(* Logix 5000 project; controller Transcat vendor 1 type 14 code 152 rev 32.11; software revision 32.02 *)

TASK MainTask (continuous, watchdog 500 ms) : MainProgram

MODULES
   Local : vendor 1 type 14 code 152 (PointIO 0, rev 32.11)
      MX201_LowerHowesVFD : PowerFlex 525-EENET (Ethernet 192.168.1.192, rev 5.1, Output RPI 20 ms)   // VFD for Lower Howes Mixer
           MX201_LowerHowesVFD:I.Ready   // LowerHowes Drive Ready Status
           MX201_LowerHowesVFD:I.Faulted   // LowerHowes Drive Faulted
           MX201_LowerHowesVFD:I.Active   // LowerHowes Drive Active
           MX201_LowerHowesVFD:O.Stop   // Drive Stop
      MX101_UpperHowesVFD : PowerFlex 525-EENET (Ethernet 192.168.1.191, rev 5.1, Output RPI 20 ms)   // VFD for Upper Howes Mixer
           MX101_UpperHowesVFD:I.Faulted   // UpperHowes Drive Faulted
           MX101_UpperHowesVFD:I.Active   // UpperHowes Drive Active
           MX101_UpperHowesVFD:I.Ready   // UpperHowes Drive Ready Status
           MX101_UpperHowesVFD:O.FreqCommand   // Input Hz into Source A: 0-60 Hz range
           MX101_UpperHowesVFD:O.Stop   // Drive Stop
           MX101_UpperHowesVFD:O.Start   // Drive Start
      VF101_Medium_Feeder : PowerFlex 525-EENET (Ethernet 192.168.1.193, rev 5.1, Output RPI 20 ms)   // Medium Feeder
      VF201_Small_Feeder_2 : PowerFlex 525-EENET (Ethernet 192.168.1.194, rev 5.1, Output RPI 20 ms)   // Small Feeder 2
      Thayer1_BS : ETHERNET-MODULE (Ethernet 192.168.1.140, rev 1.1, Output RPI 50 ms)   // Thayer 1 Weight Belt Feeder
      SBC2000_1_Acrison : ETHERNET-MODULE (Ethernet 192.168.1.150, rev 1.1, Output RPI 250 ms)   // Acrison Drive 1 to control Small Feeder 1
           SBC2000_1_Acrison:I.Data[1]   // PV - Feedrate - kg/hr
           SBC2000_1_Acrison:I.Data[2]   // Totalizer 1 - kg
           SBC2000_1_Acrison:I.Data[4]   // Hopper Level - %
           SBC2000_1_Acrison:I.Data[3]   // OT - Motor Speed - %
           SBC2000_1_Acrison:I.Data   // Ethernet Input Array
           SBC2000_1_Acrison:I.Data[0]   // SP-FeedRate - kg/hr
           SBC2000_1_Acrison:O.Data[15]   // When Command_Bits is 1, machine is running.
      Thayer2_BS : ETHERNET-MODULE (Ethernet 192.168.1.160, rev 1.1, Output RPI 50 ms)   // Thayer 2 Weigh Belt Feeder
      AENTPointIO : 1734-AENT (Ethernet 192.168.1.190, rev 3.1, Output RPI 20 ms)
         Slot1_420_8Input : vendor 1 type 115 code 210 (PointIO 1, rev 3.1, Input RPI 80 ms)
              AENTPointIO:1:I.Ch0Data   // LowerHowesSpeedSensorSignal
         Slot2_24V_8DI : 1734-IB8 (PointIO 2, rev 3.1)
      Discrete_IO : Embedded (PointIO 1, rev 32.11, Output RPI 20 ms)
           Local:1:O.Data.0   // Red Beacon Light
           Local:1:O.Data.3   // Blue Beacon Light
           Local:1:O.Data.1   // Yellow Beacon Light
           Local:1:O.Data.2   // Green Beacon Light
           Local:1:O.Data.4   // Beacon Buzzer/Sound
END_MODULES

TYPE Acrison_Feeder :   // Acrison Feeder Tags
STRUCT
   AutoMan : BOOL;   // On - Auto Control - follows AutoRun bit, Off - Manaul Control - follows Manual Run bit
   ManualRun : BOOL;   // On - Runs feeder in Manual, Off - Stops feeder in manual
   AutoRun : BOOL;   // On - Runs feeder in Auto Off - Stops feeder in Auto
   Interlock : BOOL;   // Interlock bit - if on - Feeder will not run
   Output : BOOL;   // On - Feeder runs, Off Feeder stops
   Int_Status : DINT;   // 32 Status bits from feeder
   SP_HMI : REAL;   // setpoint from HMI
   SP_READ : REAL;   // setpoint read back from controller
   Enable : BOOL;   // Enable logic to run feeder
   OT_Actual_Hz : REAL;   // The current output of the VFD in Hz
   FreqHz_Real : REAL;   // The command frequency of the drive in Hz
   CycleTime : TIMER;   // running time of current cycle
   CampTime : TIMER;   // running time of current campaign / batch
   TotalTime : TIMER;   // total time the device / motor has run since last reset
   OneShots : BOOL[32];   // 32 Booleans to hold one-shots assicated with this device
   TimeRunTarget : DINT;   // Target Amount of time in seconds to run the device
   StartDelay : TIMER;   // Delay before motor start
   StartDelayms : DINT;   // Start delay in milliseconds
   TimeRunStart : BOOL;   // Bit to start and run a timed run
END_STRUCT
END_TYPE

TYPE BronkhorstFlowMeter :   // Read and write values for Bronkhorst Flow Meters
STRUCT
   SP_R : REAL;   // Set Point - FlowRate - Read - g/min - read from Flow Meter
   PV_R : REAL;   // Process Variable - FlowRate - Read - g/min
   OT_R : REAL;   // Output - PumpSpeed - Read - %
   TempC : REAL;   // Temperaure - Read - Deg C
   Density : REAL;   // Density - Read - g/liter
   Usertag : STRING;   // User Tag in Flow Meter - String
   FBNode : INT;   // Flow Bus Node # - Integer
   Model : STRING;   // Flow Meter Model #
   Serial : STRING;   // Flow Meter Serial #
   Capacity : REAL;   // Max Flow Rate of Flow Meter
   Enable : BOOL;   // Device enable bit
   AutoMan : BOOL;   // Select Auto / Manual Mode
   AutoRun : BOOL;   // On / Off in Auto Mode
   ManualRun : BOOL;   // On / Off- in Manual Mode
   Interlock : BOOL;   // Interlock Bit
   Output : BOOL;   // Output Bit for Device
   SP_HMI : REAL;   // Setpoint from HMI
   SP_W : REAL;   // Setpoint - flowrate g/min - write to Flow Meter from PLC
   Connected : BOOL;   // Is flow meter connecte to the flow bus network
   Alarm : BOOL;   // Alarm Bit - if on flow meter in ALarm Status
   Running : BOOL;   // the flow meter is running / dosing
   AlarmReset : BOOL;   // bit to toggle to reset alarm
   AlarmID : INT;   // Integer # that describes the type of Alarm
   ReadTime : INT;   // time in milliseconds to read the flow meter data
   DevPct : REAL;   // % deviation of process variable from setpoint
   CycleTime : TIMER;   // running time of current cycle
   CampTime : TIMER;   // running time of current campaign
   TotalTime : TIMER;   // total time the device / motor has run since last reset
   OneShots : BOOL[32];   // 32 Booleans to hold one-shots assicated with this device
   TimeRunTarget : DINT;   // Target Amount of time in seconds to run the device
   StartDelay : TIMER;   // Delay before motor start
   StartDelayms : DINT;   // Start delay in milliseconds
   TimeRunStart : BOOL;   // Bit to start and run a timed run
END_STRUCT
END_TYPE

TYPE Howes_Mixer :   // Howes Mixer Tags
STRUCT
   AutoMan : BOOL;   // On - Auto Control - follows AutoRun bit, Off - Manaul Control - follows Manual Run bit
   ManualRun : BOOL;   // On - Runs feeder in Manual, Off - Stops feeder in manual
   AutoRun : BOOL;   // On - Runs feeder in Auto Off - Stops feeder in Auto
   Interlock : BOOL;   // Interlock bit - if on - Feeder will not run
   Output : BOOL;   // On - Feeder runs, Off Feeder stops
   Int_Status : DINT;   // 32 Status bits from feeder
   SP_HMI : REAL;   // setpoint from HMI
   SP_READ : REAL;   // setpoint read back from controller
   Enable : BOOL;   // Enable logic to run mixer
   FreqHz_Real : REAL;   // Frequency in Hz expressed as real #
   OT_Actual_Hz : REAL;   // The current output of the drive in Hz
   CycleTime : TIMER;   // currnet cycle run time
   CampTime : TIMER;   // current campaign run time
   TotalTime : TIMER;   // total run time since last reset
   OneShots : BOOL[32];   // 32 Booleans to hold one shots associated with this device
   TimeRunTarget : DINT;   // Target Amount of time in seconds to run the device
   TimeRunStart : BOOL;   // Bit to start and run a timed run
   StartDelay : TIMER;   // Delay before motor starts
   StartDelayms : DINT;   // Delay before motor starts in milliseconds
   RPM : REAL;   // RPM from speed sensor
END_STRUCT
END_TYPE

TYPE Thayer_WB_Feeder :   // Thayer WB Feeder Tags
STRUCT
   AutoMan : BOOL;   // On - Auto Control - follows AutoRun bit, Off - Manaul Control - follows Manual Run bit
   ManualRun : BOOL;   // On - Runs feeder in Manual, Off - Stops feeder in manual
   AutoRun : BOOL;   // On - Runs feeder in Auto Off - Stops feeder in Auto
   Interlock : BOOL;   // Interlock bit - if on - Feeder will not run
   Output : BOOL;   // On - Feeder runs, Off Feeder stops
   Int_Status : DINT;   // 32 Status bits from feeder
   SP_HMI : REAL;   // setpoint from HMI
   SP_READ : REAL;   // setpoint read back from controller
   Enable : BOOL;   // Enable logic to run feeder
   CycleTime : TIMER;   // current cycle run time
   CampTime : TIMER;   // current campaing run time
   TotalTime : TIMER;   // total run time since last reset
   OneShots : BOOL[32];   // 32 Booleans to hold one-shots assicated with this device
   TimeRunTarget : DINT;   // Target Amount of time in seconds to run the device - from recipe
   StartDelay : TIMER;   // Delay before starting motor / equipment
   StartDelayms : DINT;   // Start delay in milliseconds
   TimeRunStart : BOOL;   // Bit to start and run a timed run
END_STRUCT
END_TYPE

VAR_GLOBAL   (* controller tags *)
   AcrisonFeedRateSetPoint : MESSAGE;   // Message Command to Write to Feed Rate Set Point in Acrison from GF103.SP_HMI in kg/hr
        MessageParameters(ServiceCode := 16#0010, LocalElement := GF301.SP_HMI, ...)
   alwaysOFF : BOOL := 1;
   BeaconBeepAlarm : ALIAS FOR Local:1:O.Data.4;   // Beep Alarm
   BeaconBlueLight : ALIAS FOR Local:1:O.Data.3;   // Blue Beacon Light
   BeaconGreenLight : ALIAS FOR Local:1:O.Data.2;   // Green Beacon Light
   BeaconRedLight : ALIAS FOR Local:1:O.Data.0;   // Red Beacon Light
   BeaconYellowLight : ALIAS FOR Local:1:O.Data.1;   // Yellow Beacon Light
   Beep : BOOL;   // Bit to Activte Beacon Alarm
   FT103 : BronkhorstFlowMeter := (PV_R := -36.801758, TempC := 22.806396, Density := 9999.0, Usertag := 'FT-103', Model := 'M55-RGD-25-0-S', Serial := 'M22213015A', Capacity := 1000.00006, Enable := 1, SP_HMI := 45.67, Connected := 1, Alarm := 1, AlarmID := 40, ReadTime := 72, CycleTime.PRE := 288000000, CycleTime.ACC := 5305, CampTime.PRE := 28800000, CampTime.ACC := 10001, TotalTime.PRE := 999999999, TotalTime.ACC := 47616, StartDelay.PRE := 1000, StartDelayms := 1);
   FT104 : BronkhorstFlowMeter := (PV_R := -6.675215, TempC := 22.177925, Density := 9999.0, Usertag := 'FT-104          ', Model := 'M55-RGD-25-0-S', Serial := 'M22213015C', Capacity := 10000.0, Enable := 1, SP_HMI := 100.0, Connected := 1, ReadTime := 95, CycleTime.PRE := 288000000, CycleTime.ACC := 4100, CampTime.PRE := 28800000, CampTime.ACC := 10001, TotalTime.PRE := 999999999, TotalTime.ACC := 72384, StartDelay.PRE := 2000, StartDelayms := 2);
   FT105 : BronkhorstFlowMeter := (PV_R := 0.5933827, TempC := 29.03157, Density := 4.8631186, Usertag := 'FT-105          ', Model := 'M14-RGD-22-0-S', Serial := 'M20210127A', Capacity := 202.79999, Enable := 1, SP_HMI := 56.78, Connected := 1, ReadTime := 63, CycleTime.PRE := 288000000, CycleTime.ACC := 5050, CampTime.PRE := 28800000, CampTime.ACC := 10001, TotalTime.PRE := 999999999, TotalTime.ACC := 27737, StartDelay.PRE := 4000, StartDelayms := 4);
   GF101 : Thayer_WB_Feeder := (SP_HMI := 14.7, SP_READ := 14.6875, Enable := 1, CycleTime.PRE := 288000000, CycleTime.ACC := 2365, CampTime.PRE := 28800000, CampTime.ACC := 10001, TotalTime.PRE := 999999999, TotalTime.ACC := 1588506, StartDelay.PRE := 5000, StartDelayms := 5);   // Thayer 1 Tags
   GF201 : Thayer_WB_Feeder := (SP_HMI := 12.5, SP_READ := 12.5, Enable := 1, CycleTime.PRE := 288000000, CycleTime.ACC := 9602, CampTime.PRE := 28800000, CampTime.ACC := 10001, TotalTime.PRE := 999999999, TotalTime.ACC := 1608497, StartDelay.PRE := 3000, StartDelayms := 3);   // Thayer 2 Tags
   GF301 : Acrison_Feeder := (Int_Status := 591964, SP_HMI := 5.0, Enable := 1, CycleTime.PRE := 288000000, CycleTime.ACC := 6447, CampTime.PRE := 28800000, CampTime.ACC := 10001, TotalTime.PRE := 999999999, TotalTime.ACC := 1606494, StartDelay.PRE := 2000, StartDelayms := 2);   // GF103 - Small Feeder 1
        .Int_Status.11   // Alarm
        .Int_Status.13   // Empty
        .Int_Status.10   // Overfill / Empty
        .Int_Status.3   // SP Int-1 / Ext-0
        .Int_Status   // 32 Bit Status Int
        .Int_Status.0   // Run-1 / Stop-0
        .Int_Status.5   // Batch-1 / Cont-0
        .Int_Status.4   // Mode - Grav-1 / Vol-0
        .Int_Status.6   // Batch Complete
        .Int_Status.1   // Refil
        .Int_Status.7   // Bribble
        .Int_Status.12   // Message
        .Int_Status.9   // Low Level
        .Int_Status.14   // Overfill
        .Int_Status.15   // Acrilock
        .Int_Status.16   // No Scale
        .Int_Status.17   // Deviation
        .Output   // GF103 - Acrison Small Feeder Run Bit
        .Int_Status.2   // AutoRefill
        .Int_Status.8   // High Level
   GreenFlashingOff : TIMER := (PRE := 500);
   GreenFlashingOn : TIMER := (PRE := 500);
   HertzSetting : ALIAS FOR MX101_UpperHowesVFD:O.FreqCommand.0;   // UserHzSetting
   MSG_FROM_SLC500 : INT[10] := ([1] := 2500, [2] := 200, [3] := 300, [4] := 400, [5] := 500, [6] := 16, [7] := 17, [8] := 18, [9] := 19); {produced}
   MX101 : Howes_Mixer := (SP_HMI := 5.0, Enable := 1, FreqHz_Real := 3.0, CycleTime.PRE := 288000000, CycleTime.ACC := 3118, CampTime.PRE := 28800000, CampTime.ACC := 10001, TotalTime.PRE := 999999999, TotalTime.ACC := 1718665, StartDelay.PRE := 5000, StartDelayms := 5);
   MX201 : Howes_Mixer := (SP_HMI := 10.0, Enable := 1, FreqHz_Real := 6.0, CycleTime.PRE := 28800000, CycleTime.ACC := 7089, CampTime.PRE := 28800000, CampTime.ACC := 10001, TotalTime.PRE := 999999999, TotalTime.ACC := 835800, StartDelay.PRE := 2000, StartDelayms := 2, RPM := -0.04);
   PowerOffThayer1 : BOOL;
   PowerOnThayer1 : BOOL;
   RandomFloat : REAL[20] := ([1] := 7.316811, [2] := 20.713356, [3] := 16.079597, [4] := 74.3938, [5] := 86.28061, [6] := 69.73996, [7] := 47.361, [8] := 43.876316, [9] := 89.62069, [10] := 56.526745);
   RecipeStart : BOOL;   // Bit to start and stop a recipe execution
   StartBeepTimer : TIMER := (PRE := 2500);   // Timer to sound the beep alarm before starting a device
   TempReal1 : REAL;
   Thayer1_SP : REAL := 20.0;
   Thayer1Ackn_SilenceRequest : BOOL;
   Thayer1Automatic : BOOL;
   Thayer1Data : REAL[40] := ([0] := -0.072265625, [1] := 4.6216e-41, [3] := 14.6875, [4] := 2.0, [9] := -0.19335938, [10] := -0.19343926, [11] := 7.512e-42, [15] := -0.071777344, [16] := 70.84617, [17] := 1.6071e-41, [19] := -0.072265625);
        [10]   // Totalizer 2
        [3]   // SetPoint
        [2]   // Running Speed
        [0]   // Running Load
        [1]   // Running Rate
        [9]   // Totalizer 1
   Thayer1PowerOn : BOOL;
   Thayer1ResetTotalizers : BOOL;
   Thayer1SetPoint : REAL[1];
   Thayer1SpeedControl : REAL := 20.0;
   Thayer2_SP : REAL := 20.0;
   Thayer2Automatic : BOOL;
   Thayer2Data : REAL[40] := ([0] := 3.609375, [1] := 7.6406e-41, [3] := 12.5, [15] := 3.609375, [16] := 70.91538, [17] := 1.6071e-41, [19] := 3.609375);
   Thayer2PowerOn : BOOL;
   Thayer2ResetTotalizers : BOOL;
   Thayer2SpeedControl : REAL := 20.0;
   UHStartOneShot : BOOL;
   UHStopOneShot : BOOL;
   UpHowesHMIRun : BOOL;
   UpHowesHMIStop : BOOL;
   UpHowesSpeedHMI : INT;
   UpperHowesSpeed : INT := 2500;
   UpperHowesStart : BOOL;
   UpperHowesStop : BOOL;
   VF101 : Acrison_Feeder := (SP_HMI := 10.0, Enable := 1, FreqHz_Real := 6.0, CycleTime.PRE := 288000000, CycleTime.ACC := 7359, CampTime.PRE := 28800000, CampTime.ACC := 10001, TotalTime.PRE := 999999999, TotalTime.ACC := 1720239, StartDelay.PRE := 5000, StartDelayms := 5);   // Medium Feeder Tags
   VF201 : Acrison_Feeder := (SP_HMI := 10.0, Enable := 1, FreqHz_Real := 6.0, CycleTime.PRE := 288000000, CycleTime.ACC := 13534, CampTime.PRE := 28800000, CampTime.ACC := 10001, TotalTime.PRE := 999999999, TotalTime.ACC := 1964985, StartDelay.PRE := 5000, StartDelayms := 5);   // Small Feeder 2 Tags
   YellowFlashOff : TIMER := (PRE := 500);
   YellowFlashOn : TIMER := (PRE := 500);
END_VAR

PROGRAM MainProgram   (* main routine MainRoutine *)
VAR
   AcrisonSpeedControl : REAL := 1.0;
   AcrisonSpeedControl2 : REAL := 15.0;
   Command_Bits : INT;
        .0   // GF103 - Acrison Small Feeder 1 - Run/Stop
   HertzInput : INT := 20;
   Int_Status : DINT := 540252;
   LowerHowesSpeedSensor : REAL := -74.39945;
   PowerOffACrison : BOOL := 1;
   PowerOnAcrison : BOOL;
   SCL_01 : SCALE := (In := -3.0, InRawMax := 16384.0, InRawMin := 3271.0, InEUMax := 300.0, Out := -74.90277, MinAlarm := 1);
   SCL_02 : SCALE := (In := 19.0, InRawMax := 16384.0, InRawMin := 3271.0, InEUMax := 300.0, Out := -74.39945, MinAlarm := 1);
   SpeedSensorUpperHowesSpeed : REAL := -74.90277;
   T1 : TIMER := (PRE := 10000);
   T2 : TIMER := (PRE := 10000, ACC := 10000, EN := 1, DN := 1);
END_VAR

ROUTINE FT103_Oil_Dosing   (* ladder *)
// Logic to control FT103
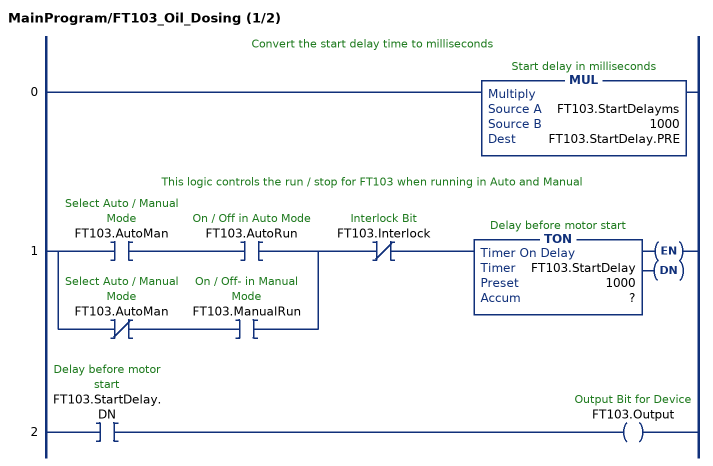
   // Convert the start delay time to milliseconds
   0: MUL(FT103.StartDelayms,1000,FT103.StartDelay.PRE);
   // This logic controls the run / stop for FT103 when running in Auto and Manual
   1: [XIC(FT103.AutoMan) XIC(FT103.AutoRun) ,XIO(FT103.AutoMan) XIC(FT103.ManualRun) ]XIO(FT103.Interlock)TON(FT103.StartDelay,?,?);
   2: XIC(FT103.StartDelay.DN)OTE(FT103.Output);
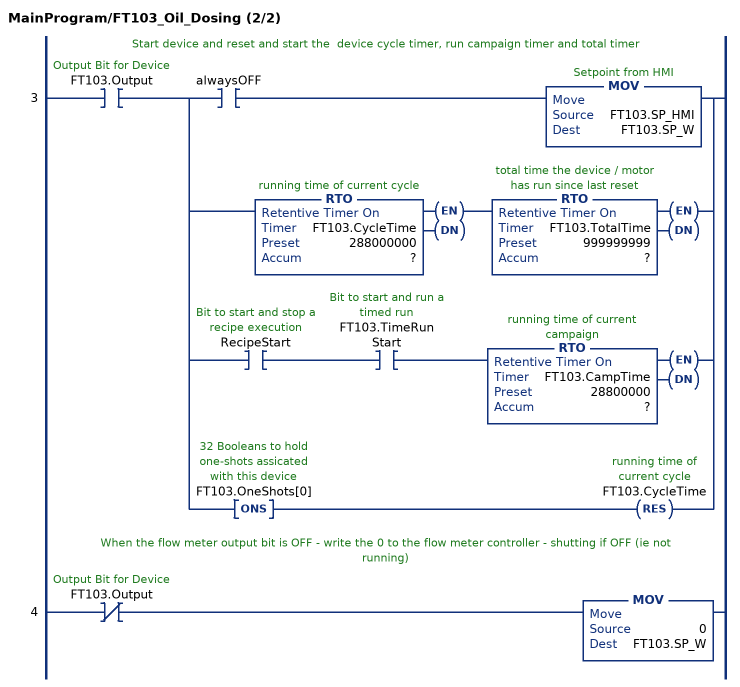
   // Start device and reset and start the  device cycle timer, run campaign timer and total timer
   3: XIC(FT103.Output)[XIC(alwaysOFF) MOV(FT103.SP_HMI,FT103.SP_W) ,[RTO(FT103.CycleTime,?,?) RTO(FT103.TotalTime,?,?) ,XIC(RecipeStart) XIC(FT103.TimeRunStart) RTO(FT103.CampTime,?,?) ,ONS(FT103.OneShots[0]) RES(FT103.CycleTime) ] ];
   // When the flow meter output bit is OFF - write the 0 to the flow meter controller - shutting if OFF (ie not running)
   4: XIO(FT103.Output)MOV(0,FT103.SP_W);
END_ROUTINE

ROUTINE FT104_Water_Dosing   (* ladder *)
// FT104 Control Logic
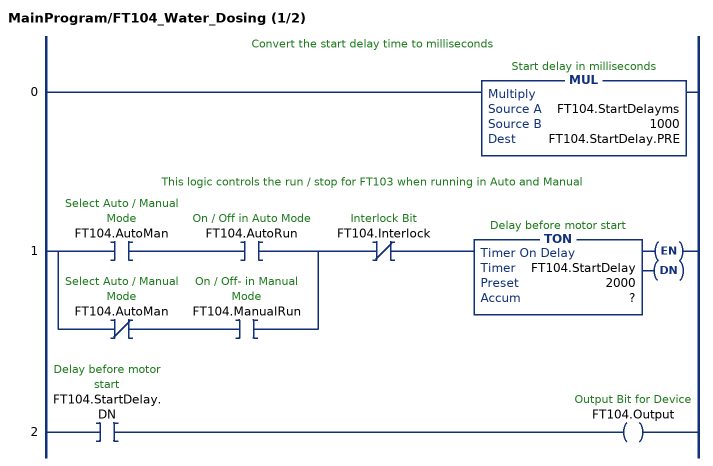
   // Convert the start delay time to milliseconds
   0: MUL(FT104.StartDelayms,1000,FT104.StartDelay.PRE);
   // This logic controls the run / stop for FT103 when running in Auto and Manual
   1: [XIC(FT104.AutoMan) XIC(FT104.AutoRun) ,XIO(FT104.AutoMan) XIC(FT104.ManualRun) ]XIO(FT104.Interlock)TON(FT104.StartDelay,?,?);
   2: XIC(FT104.StartDelay.DN)OTE(FT104.Output);
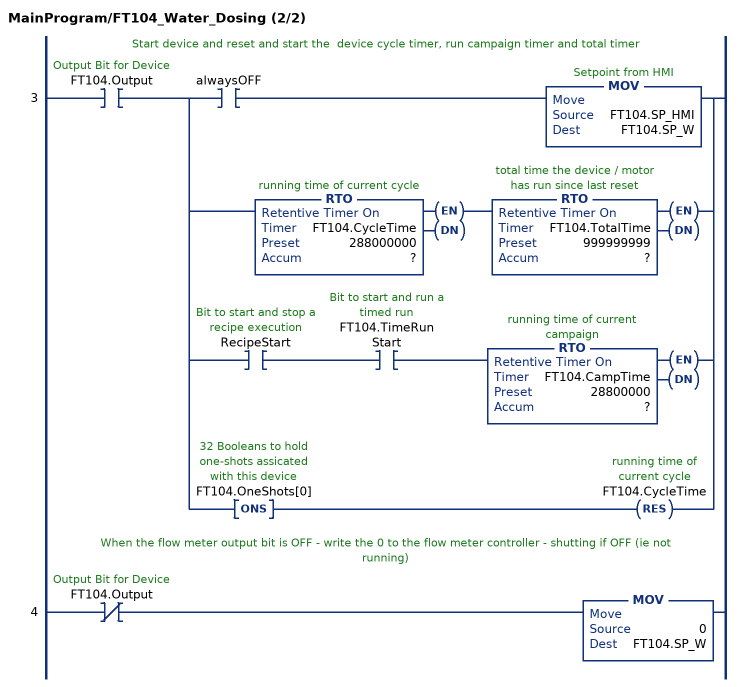
   // Start device and reset and start the  device cycle timer, run campaign timer and total timer
   3: XIC(FT104.Output)[XIC(alwaysOFF) MOV(FT104.SP_HMI,FT104.SP_W) ,[RTO(FT104.CycleTime,?,?) RTO(FT104.TotalTime,?,?) ,XIC(RecipeStart) XIC(FT104.TimeRunStart) RTO(FT104.CampTime,?,?) ,ONS(FT104.OneShots[0]) RES(FT104.CycleTime) ] ];
   // When the flow meter output bit is OFF - write the 0 to the flow meter controller - shutting if OFF (ie not running)
   4: XIO(FT104.Output)MOV(0,FT104.SP_W);
END_ROUTINE

ROUTINE FT105_Fragrance_Dosing   (* ladder *)
// FT105 Control Logic
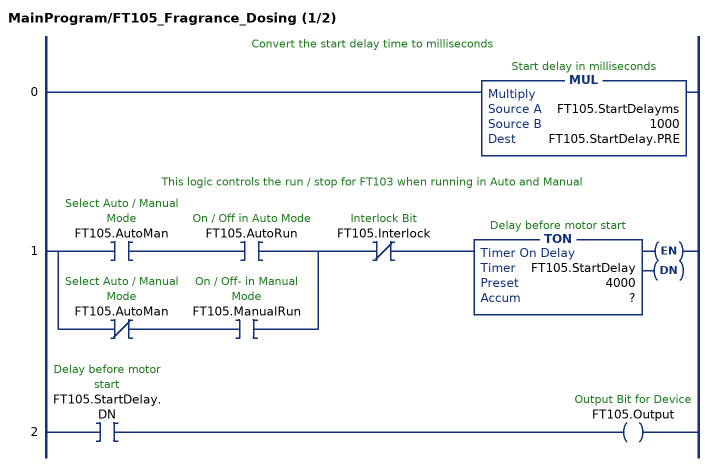
   // Convert the start delay time to milliseconds
   0: MUL(FT105.StartDelayms,1000,FT105.StartDelay.PRE);
   // This logic controls the run / stop for FT103 when running in Auto and Manual
   1: [XIC(FT105.AutoMan) XIC(FT105.AutoRun) ,XIO(FT105.AutoMan) XIC(FT105.ManualRun) ]XIO(FT105.Interlock)TON(FT105.StartDelay,?,?);
   2: XIC(FT105.StartDelay.DN)OTE(FT105.Output);
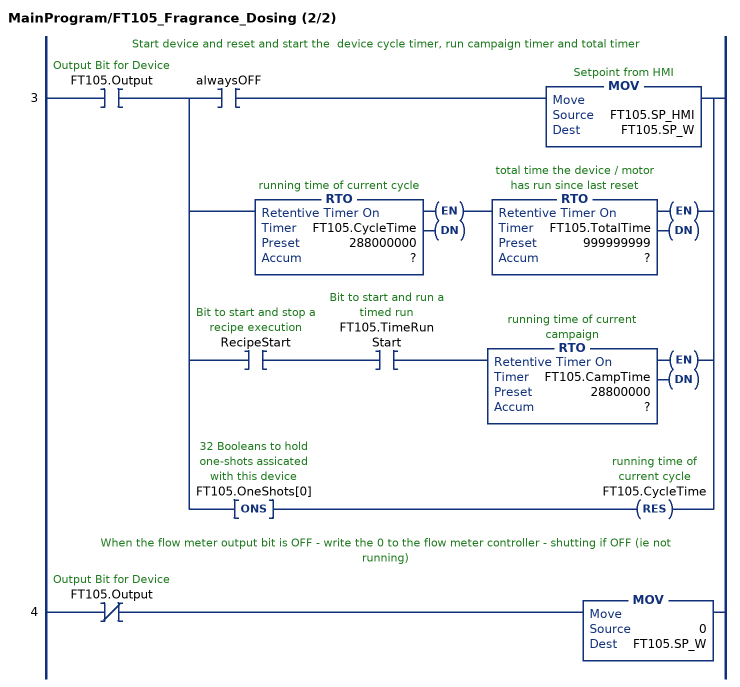
   // Start device and reset and start the  device cycle timer, run campaign timer and total timer
   3: XIC(FT105.Output)[XIC(alwaysOFF) MOV(FT105.SP_HMI,FT105.SP_W) ,[RTO(FT105.CycleTime,?,?) RTO(FT105.TotalTime,?,?) ,XIC(RecipeStart) XIC(FT105.TimeRunStart) RTO(FT105.CampTime,?,?) ,ONS(FT105.OneShots[0]) RES(FT105.CycleTime) ] ];
   // When the flow meter output bit is OFF - write the 0 to the flow meter controller - shutting if OFF (ie not running)
   4: XIO(FT105.Output)MOV(0,FT105.SP_W);
END_ROUTINE

ROUTINE GF101_Thayer1_WB_Feeder   (* ladder *)
// Thayer1 WB Feeder Control Logic (Old Limestone Feeder)
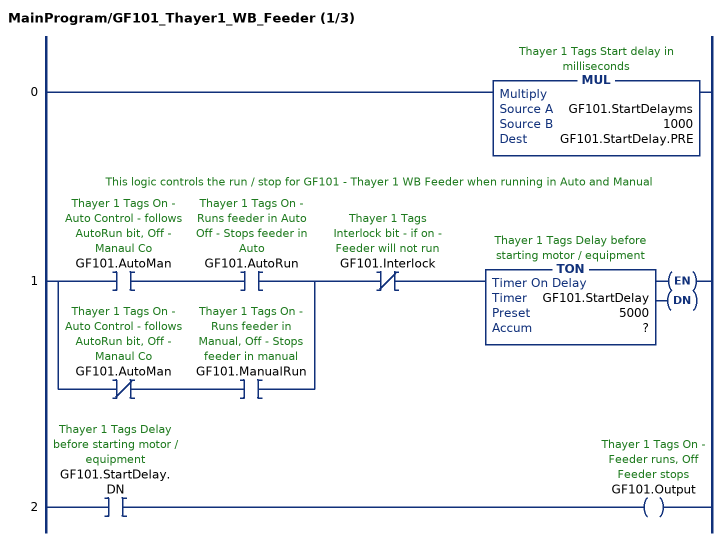
   0: MUL(GF101.StartDelayms,1000,GF101.StartDelay.PRE);
   // This logic controls the run / stop for GF101 - Thayer 1 WB Feeder when running in Auto and Manual
   1: [XIC(GF101.AutoMan) XIC(GF101.AutoRun) ,XIO(GF101.AutoMan) XIC(GF101.ManualRun) ]XIO(GF101.Interlock)TON(GF101.StartDelay,?,?);
   2: XIC(GF101.StartDelay.DN)OTE(GF101.Output);
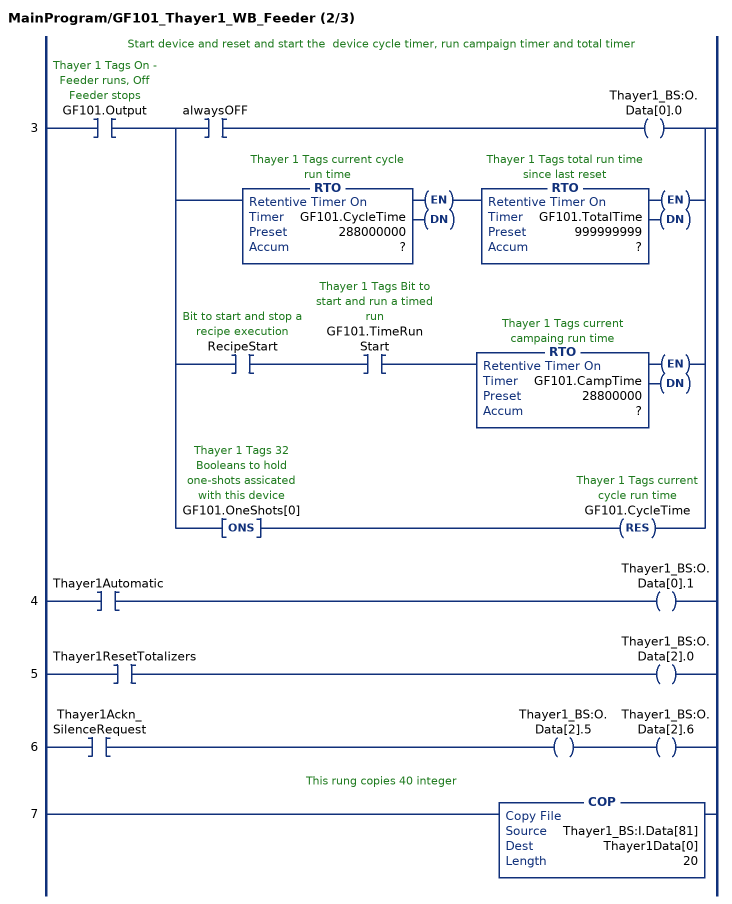
   // Start device and reset and start the  device cycle timer, run campaign timer and total timer
   3: XIC(GF101.Output)[XIC(alwaysOFF) OTE(Thayer1_BS:O.Data[0].0) ,[RTO(GF101.CycleTime,?,?) RTO(GF101.TotalTime,?,?) ,XIC(RecipeStart) XIC(GF101.TimeRunStart) RTO(GF101.CampTime,?,?) ,ONS(GF101.OneShots[0]) RES(GF101.CycleTime) ] ];
   4: XIC(Thayer1Automatic)OTE(Thayer1_BS:O.Data[0].1);
   5: XIC(Thayer1ResetTotalizers)OTE(Thayer1_BS:O.Data[2].0);
   6: XIC(Thayer1Ackn_SilenceRequest)OTE(Thayer1_BS:O.Data[2].5)OTE(Thayer1_BS:O.Data[2].6);
   // This rung copies 40 integer
   7: COP(Thayer1_BS:I.Data[81],Thayer1Data[0],20);
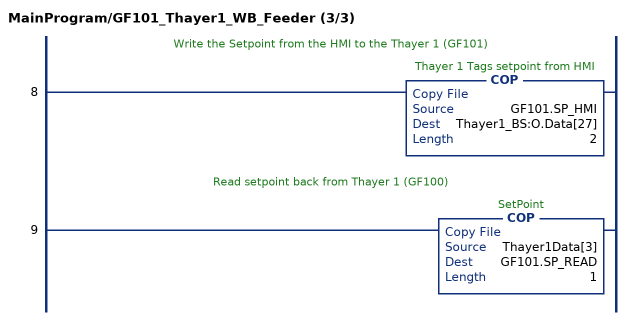
   // Write the Setpoint from the HMI to the Thayer 1 (GF101)
   8: COP(GF101.SP_HMI,Thayer1_BS:O.Data[27],2);
   // Read setpoint back from Thayer 1 (GF100)
   9: COP(Thayer1Data[3],GF101.SP_READ,1);
END_ROUTINE

ROUTINE GF201_Thayer2_WB_Feeder   (* ladder *)
// Thayer2 WB Feeder Control Logic (Old - Bentonite Feeder)
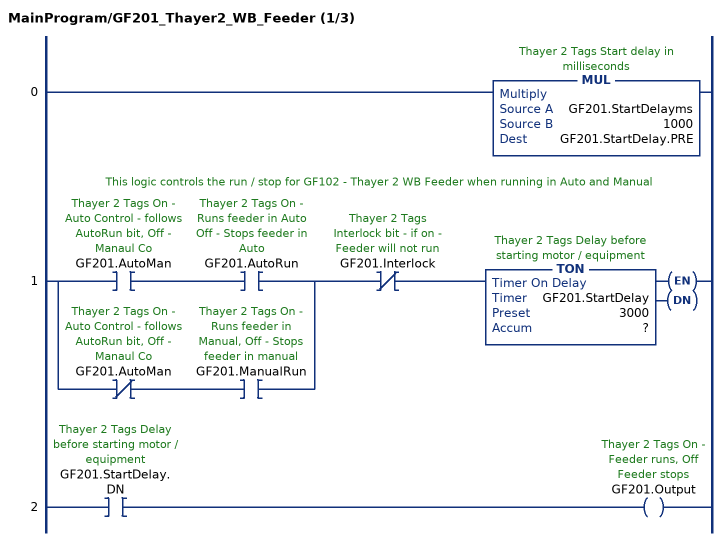
   0: MUL(GF201.StartDelayms,1000,GF201.StartDelay.PRE);
   // This logic controls the run / stop for GF102 - Thayer 2 WB Feeder when running in Auto and Manual
   1: [XIC(GF201.AutoMan) XIC(GF201.AutoRun) ,XIO(GF201.AutoMan) XIC(GF201.ManualRun) ]XIO(GF201.Interlock)TON(GF201.StartDelay,?,?);
   2: XIC(GF201.StartDelay.DN)OTE(GF201.Output);
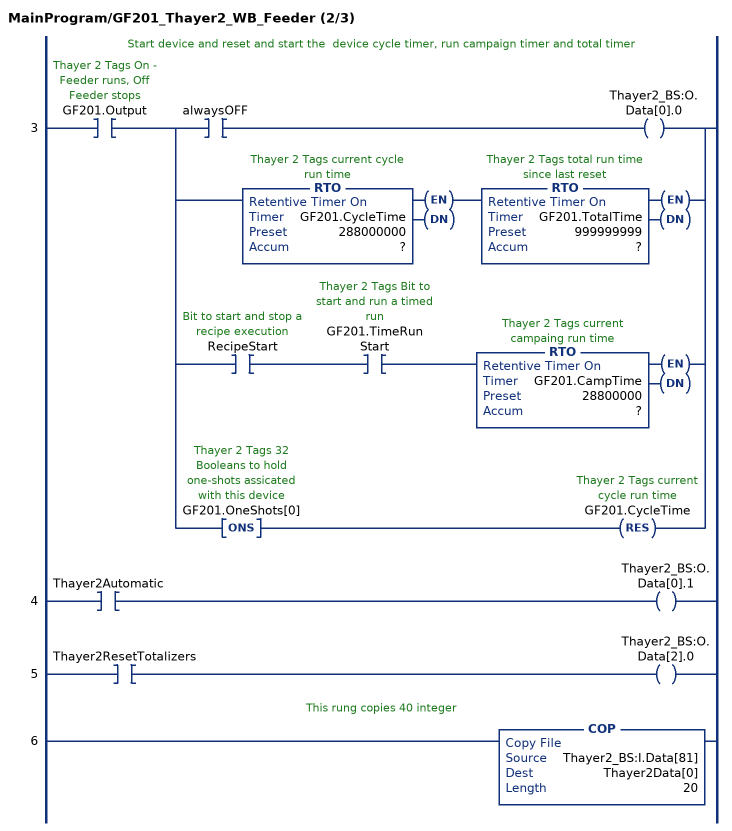
   // Start device and reset and start the  device cycle timer, run campaign timer and total timer
   3: XIC(GF201.Output)[XIC(alwaysOFF) OTE(Thayer2_BS:O.Data[0].0) ,[RTO(GF201.CycleTime,?,?) RTO(GF201.TotalTime,?,?) ,XIC(RecipeStart) XIC(GF201.TimeRunStart) RTO(GF201.CampTime,?,?) ,ONS(GF201.OneShots[0]) RES(GF201.CycleTime) ] ];
   4: XIC(Thayer2Automatic)OTE(Thayer2_BS:O.Data[0].1);
   5: XIC(Thayer2ResetTotalizers)OTE(Thayer2_BS:O.Data[2].0);
   // This rung copies 40 integer
   6: COP(Thayer2_BS:I.Data[81],Thayer2Data[0],20);
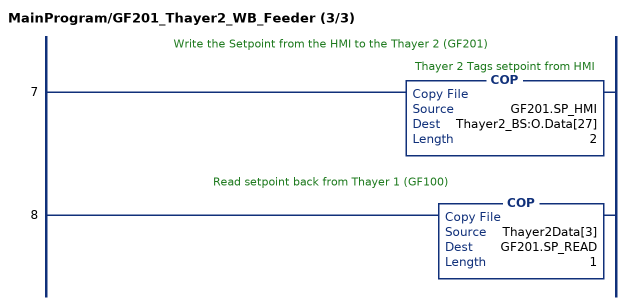
   // Write the Setpoint from the HMI to the Thayer 2 (GF201)
   7: COP(GF201.SP_HMI,Thayer2_BS:O.Data[27],2);
   // Read setpoint back from Thayer 1 (GF100)
   8: COP(Thayer2Data[3],GF201.SP_READ,1);
END_ROUTINE

ROUTINE GF301_Small_Feeder_AcrisonLIW   (* ladder *)
// Small Feeder 1 Control via Acrison Drive SBC 2000
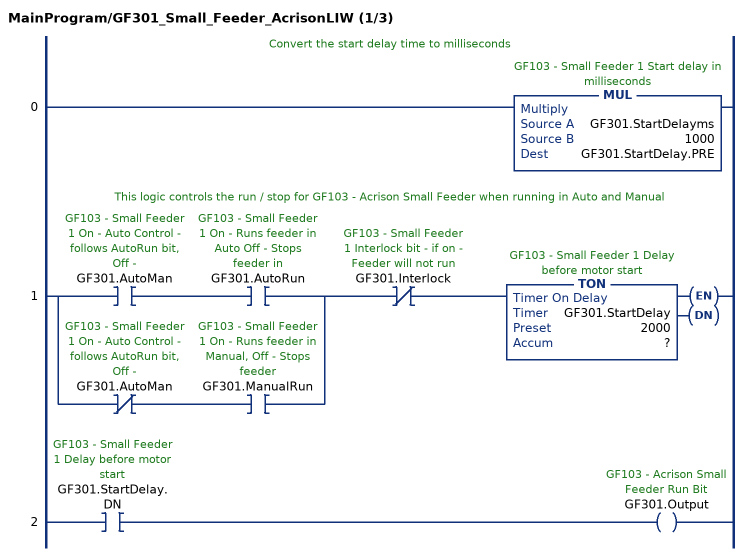
   // Convert the start delay time to milliseconds
   0: MUL(GF301.StartDelayms,1000,GF301.StartDelay.PRE);
   // This logic controls the run / stop for GF103 - Acrison Small Feeder when running in Auto and Manual
   1: [XIC(GF301.AutoMan) XIC(GF301.AutoRun) ,XIO(GF301.AutoMan) XIC(GF301.ManualRun) ]XIO(GF301.Interlock)TON(GF301.StartDelay,?,?);
   2: XIC(GF301.StartDelay.DN)OTE(GF301.Output);
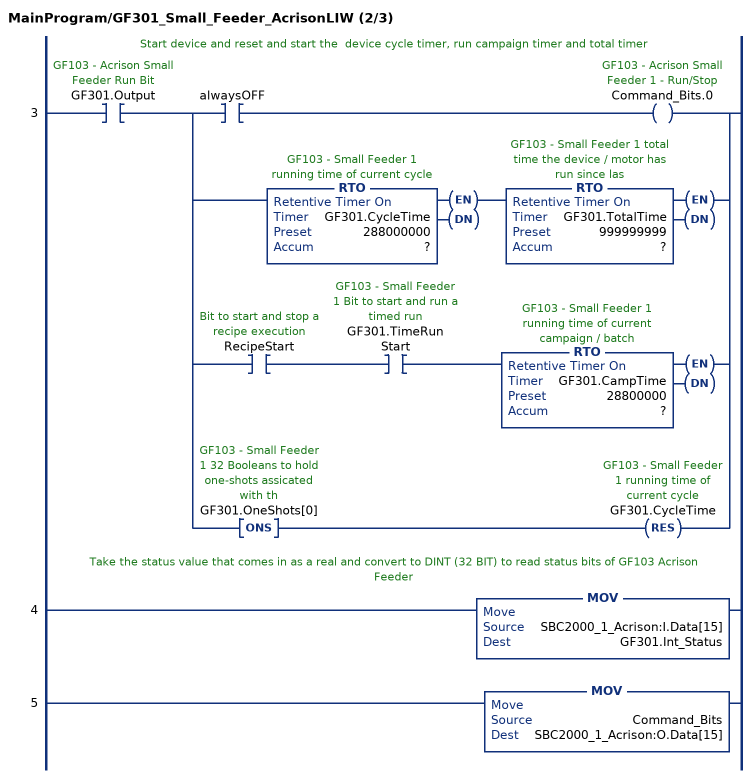
   // Start device and reset and start the  device cycle timer, run campaign timer and total timer
   3: XIC(GF301.Output)[XIC(alwaysOFF) OTE(Command_Bits.0) ,[RTO(GF301.CycleTime,?,?) RTO(GF301.TotalTime,?,?) ,XIC(RecipeStart) XIC(GF301.TimeRunStart) RTO(GF301.CampTime,?,?) ,ONS(GF301.OneShots[0]) RES(GF301.CycleTime) ] ];
   // Take the status value that comes in as a real and convert to DINT (32 BIT) to read status bits of GF103 Acrison Feeder
   4: MOV(SBC2000_1_Acrison:I.Data[15],GF301.Int_Status);
   5: MOV(Command_Bits,SBC2000_1_Acrison:O.Data[15]);
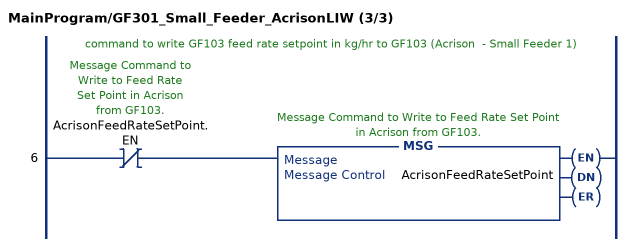
   // command to write GF103 feed rate setpoint in kg/hr to GF103 (Acrison  - Small Feeder 1)
   6: XIO(AcrisonFeedRateSetPoint.EN)MSG(AcrisonFeedRateSetPoint);
END_ROUTINE

ROUTINE Light_Beacon   (* ladder *)
// Indicator Light Beacon
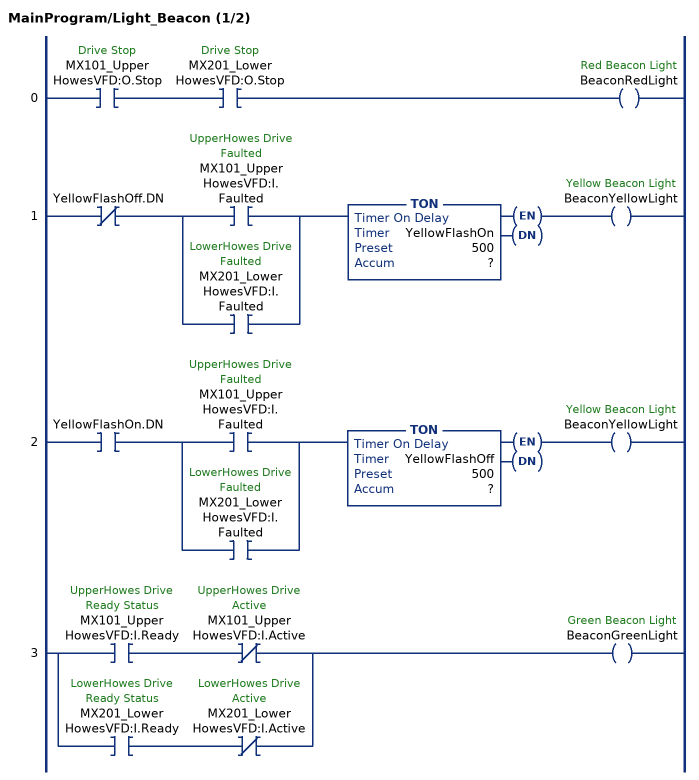
   0: XIC(MX101_UpperHowesVFD:O.Stop)XIC(MX201_LowerHowesVFD:O.Stop)OTE(BeaconRedLight);
   1: XIO(YellowFlashOff.DN)[XIC(MX101_UpperHowesVFD:I.Faulted) ,XIC(MX201_LowerHowesVFD:I.Faulted) ]TON(YellowFlashOn,?,?)OTE(BeaconYellowLight);
   2: XIC(YellowFlashOn.DN)[XIC(MX101_UpperHowesVFD:I.Faulted) ,XIC(MX201_LowerHowesVFD:I.Faulted) ]TON(YellowFlashOff,?,?)OTE(BeaconYellowLight);
   3: [XIC(MX101_UpperHowesVFD:I.Ready) XIO(MX101_UpperHowesVFD:I.Active) ,XIC(MX201_LowerHowesVFD:I.Ready) XIO(MX201_LowerHowesVFD:I.Active) ]OTE(BeaconGreenLight);
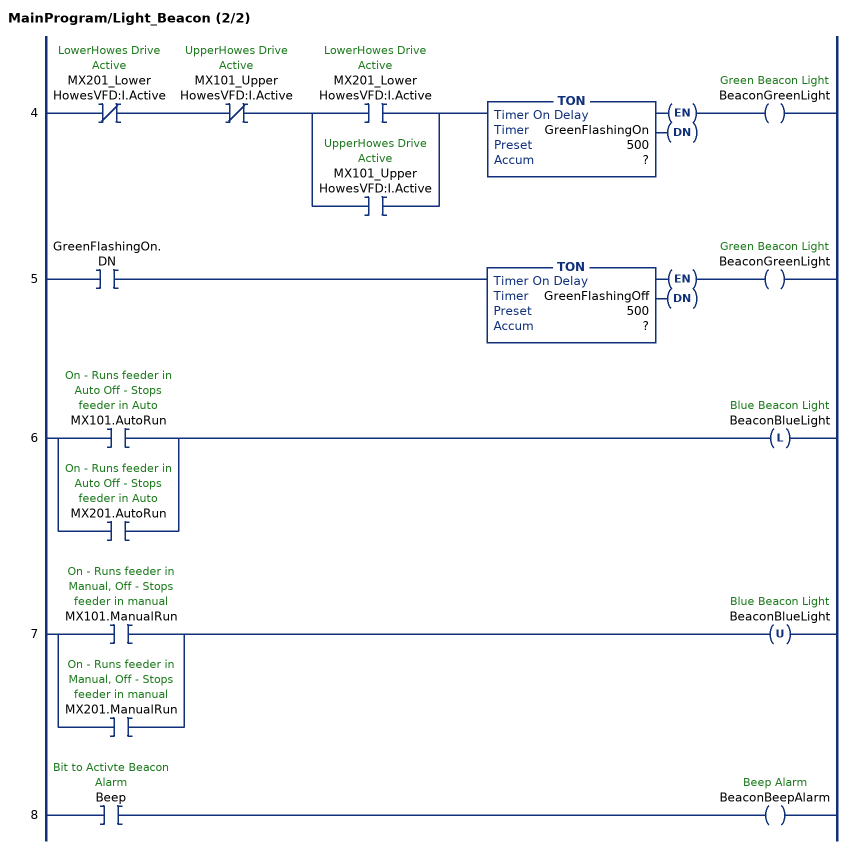
   4: XIO(MX201_LowerHowesVFD:I.Active)XIO(MX101_UpperHowesVFD:I.Active)[XIC(MX201_LowerHowesVFD:I.Active) ,XIC(MX101_UpperHowesVFD:I.Active) ]TON(GreenFlashingOn,?,?)OTE(BeaconGreenLight);
   5: XIC(GreenFlashingOn.DN)TON(GreenFlashingOff,?,?)OTE(BeaconGreenLight);
   6: [XIC(MX101.AutoRun) ,XIC(MX201.AutoRun) ]OTL(BeaconBlueLight);
   7: [XIC(MX101.ManualRun) ,XIC(MX201.ManualRun) ]OTU(BeaconBlueLight);
   8: XIC(Beep)OTE(BeaconBeepAlarm);
END_ROUTINE

ROUTINE LowerHowesSpeedScaling   (* function block diagram *)
// Lower Howes Speed Sensor 4-20 mA signal
   SHEET 1
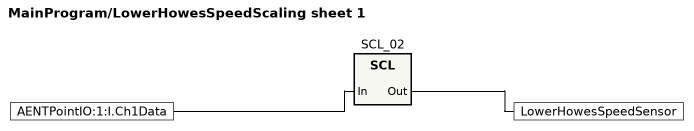
   SCL_02 : SCL(In := AENTPointIO:1:I.Ch1Data);
   LowerHowesSpeedSensor := SCL_02.Out;
END_ROUTINE
